PROGRAM MAIN 
VAR
END_VAR

SavePersistentVariables ();

END_PROGRAM

(* stored: Version 1.1.0.1, ProductVersion 3.1.4024.3
   POU MAIN: Id {89dc724e-e8f7-4f0a-8ccf-d584989e3263}, SpecialFunc None *)
